Universal Robots PolyScope program: Mycobot.urp

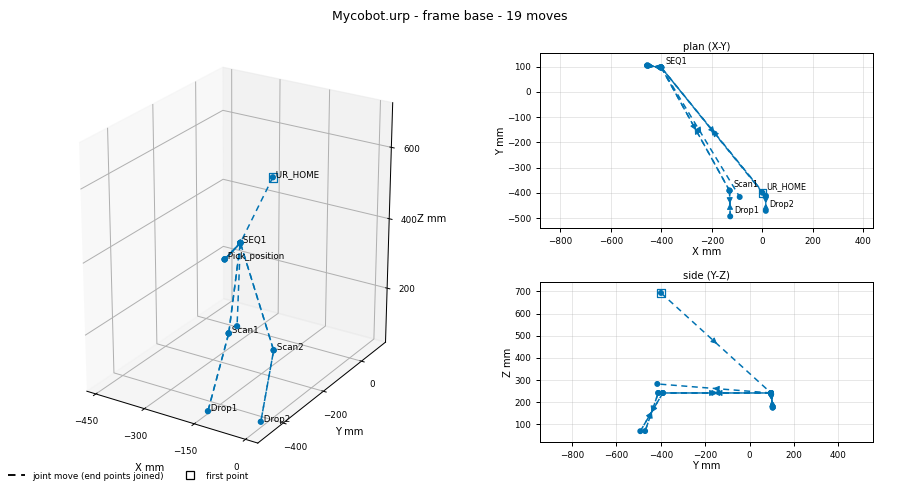
[picture p0: tool path of Mycobot.urp in frame base, 19 of 19 moves have a stored position in this frame; points joined in program order, loops and branches not executed]
Program Mycobot (installation=default directory=/programs createdIn=5.13.0 lastSavedIn=5.13.0 robotSerialNumber=20185300461)
Calibrated DH parameters: a=[-0.000193, -0.207022, -0.182437, 0.000132, -0.000092, 0]; d=[0.151833, 39.901235, 24.993935, -64.763969, 0.085421, 0.09218]; alpha=[1.57101, -0.003228, 0.001706, 1.571505, -1.572476, 0]; deltaTheta=[0, -0.556568, 7.385156, -0.545397, -0.000002, 0]
InitVariablesNode
Robot Program (runOnlyOnce=false)
  MoveJ speed 60 deg/s, acceleration 80 deg/s^2 (useActiveTCP=true) feature=Base
    Waypoint UR_HOME: TCP in base x=0.281 y=-399.322 z=693.096 mm, rx=-0.0014 ry=2.225 rz=-2.2166 rad; joints [-0.001, -90.001, 0, -89.999, 0.001, 0.001] deg; TCP offset x=0 y=0 z=175 mm, rx=0 ry=0 rz=0 rad
    Waypoint SEQ1: TCP in base x=-400.455 y=96.867 z=242.077 mm, rx=-2.2115 ry=-2.1405 rz=0.0251 rad; joints [-173.349, -123.94, -11.31, -131.69, 87.509, 8.47] deg; TCP offset x=0 y=0 z=175 mm, rx=0 ry=0 rz=0 rad
    Wait Sleep waitTime=5
    Waypoint Pick_position: TCP in base x=-456.138 y=104.432 z=176.635 mm, rx=-3.123 ry=0.1229 rz=0.0643 rad; joints [-175.863, -135.405, -11.262, -120.992, 88.708, 98.607] deg
    URCap Gripper (Robotiq_Grippers, Robotiq Inc.) dataModel(position=52.94117647058823, force=36.60130718954249, speed=10.893246187363836, positionInDouble=52.94117647058823, forceInDouble=36.60130718954249, speedInDouble=10.893246187363836, slaveIds=[9], blocking=true, robotCompliant=false)
    URCap Grip Check (Robotiq_Grippers, Robotiq Inc.) dataModel(DimensionKey=100.0, DimensionDimensionPositiveGapKey=5.0, DimensionNegativeGapKey=5.0, GripperIdKey=1, ModelDefinedKey=true, ObjectDetectedKey=true, DimensionValidationKey=false); state(isChildrenLocked=true)
      URCap If (Robotiq_Grippers, Robotiq Inc.)
        Waypoint Waypoint_1: TCP in base x=-400.458 y=96.877 z=242.084 mm, rx=-2.2115 ry=-2.1404 rz=0.0251 rad; joints [-173.351, -123.94, -11.307, -131.691, 87.509, 8.47] deg; TCP offset x=0 y=0 z=175 mm, rx=0 ry=0 rz=0 rad
      URCap Else (Robotiq_Grippers, Robotiq Inc.)
        Wait Sleep waitTime=10
        Popup Message (haltProgram=false message=NO LEGO DETECTED inputType=Text)
    Waypoint Safe_above_pik2: TCP in base x=-400.455 y=96.891 z=242.08 mm, rx=-2.2116 ry=-2.1404 rz=0.0251 rad; joints [-173.353, -123.94, -11.31, -131.689, 87.509, 8.471] deg; TCP offset x=0 y=0 z=175 mm, rx=0 ry=0 rz=0 rad
    Waypoint Scan1: TCP in base x=-130.159 y=-390.915 z=242.077 mm, rx=-0.1811 ry=-3.0992 rz=0.0857 rad; joints [-88.166, -123.94, -11.311, -131.689, 87.507, 8.471] deg; TCP offset x=0 y=0 z=175 mm, rx=0 ry=0 rz=0 rad
    Wait Sleep waitTime=3
    Waypoint Drop1: TCP in base x=-127.488 y=-492.684 z=69.679 mm, rx=-0.1841 ry=-3.0975 rz=0.0473 rad; joints [-88.165, -171.493, 34.819, -131.686, 87.506, 8.471] deg; TCP offset x=0 y=0 z=175 mm, rx=0 ry=0 rz=0 rad
    URCap Gripper (Robotiq_Grippers, Robotiq Inc.) dataModel(position=40.0, force=36.60130718954249, speed=10.893246187363836, positionInDouble=40.0, forceInDouble=36.60130718954249, speedInDouble=10.893246187363836, slaveIds=[9], blocking=true, robotCompliant=false)
    Wait Sleep waitTime=1
    Waypoint Return0: TCP in base x=-130.177 y=-390.911 z=242.06 mm, rx=-0.1811 ry=-3.0991 rz=0.0856 rad; joints [-88.166, -123.941, -11.312, -131.69, 87.503, 8.471] deg; TCP offset x=0 y=0 z=175 mm, rx=0 ry=0 rz=0 rad
    URCap Gripper (Robotiq_Grippers, Robotiq Inc.) dataModel(position=19.607843137254903, force=36.60130718954249, speed=10.893246187363836, positionInDouble=19.607843137254903, forceInDouble=36.60130718954249, speedInDouble=10.893246187363836, slaveIds=[9], blocking=true, robotCompliant=false)
    Waypoint scan01: TCP in base x=-130.136 y=-390.929 z=242.057 mm, rx=-0.1809 ry=-3.0991 rz=0.0856 rad; joints [-88.161, -123.942, -11.311, -131.689, 87.505, 8.47] deg; TCP offset x=0 y=0 z=175 mm, rx=0 ry=0 rz=0 rad
    URCap Gripper (Robotiq_Grippers, Robotiq Inc.) dataModel(position=0.0, force=36.60130718954249, speed=10.893246187363836, positionInDouble=0.0, forceInDouble=36.60130718954249, speedInDouble=10.893246187363836, slaveIds=[9], blocking=true, robotCompliant=false)
    Waypoint SEQ2: TCP in base x=-400.462 y=96.851 z=242.093 mm, rx=-2.2115 ry=-2.1404 rz=0.0252 rad; joints [-173.348, -123.938, -11.309, -131.69, 87.51, 8.472] deg; TCP offset x=0 y=0 z=175 mm, rx=0 ry=0 rz=0 rad
    Wait Sleep waitTime=5
    Waypoint Pickv2: TCP in base x=-456.135 y=104.44 z=176.645 mm, rx=-3.123 ry=0.1229 rz=0.0643 rad; joints [-175.863, -135.404, -11.261, -120.993, 88.707, 98.607] deg; TCP offset x=0 y=0 z=175 mm, rx=0 ry=0 rz=0 rad
    URCap Gripper (Robotiq_Grippers, Robotiq Inc.) dataModel(position=52.94117647058823, force=36.60130718954249, speed=10.893246187363836, positionInDouble=52.94117647058823, forceInDouble=36.60130718954249, speedInDouble=10.893246187363836, slaveIds=[9], blocking=true, robotCompliant=false)
    URCap Grip Check (Robotiq_Grippers, Robotiq Inc.) dataModel(ObjectDetectedKey=true, DimensionValidationKey=false, DimensionKey=100.0, DimensionDimensionPositiveGapKey=5.0, DimensionNegativeGapKey=5.0, GripperIdKey=1, ModelDefinedKey=true); state(isChildrenLocked=true)
      URCap If (Robotiq_Grippers, Robotiq Inc.)
        Waypoint Waypoint_2: TCP in base x=-400.465 y=96.868 z=242.087 mm, rx=-2.2115 ry=-2.1404 rz=0.0252 rad; joints [-173.35, -123.939, -11.31, -131.688, 87.51, 8.469] deg; TCP offset x=0 y=0 z=175 mm, rx=0 ry=0 rz=0 rad
      URCap Else (Robotiq_Grippers, Robotiq Inc.)
        Popup Message (haltProgram=false message=NO LEGO DETECTED inputType=Text)
    Waypoint Scan2: TCP in base x=13.397 y=-411.795 z=242.108 mm, rx=0.3685 ry=-3.0926 rz=0.0947 rad; joints [-67.888, -123.936, -11.31, -131.687, 87.509, 8.47] deg; TCP offset x=0 y=0 z=175 mm, rx=0 ry=0 rz=0 rad
    Wait Sleep waitTime=3
    Waypoint Drop2: motionParameters(nextMotionTime=4); TCP in base x=13.429 y=-470.86 z=70.27 mm, rx=0.1151 ry=-3.0804 rz=-0.1175 rad; joints [-71.076, -136.443, -37.095, -101.486, 88.026, 14.753] deg; TCP offset x=0 y=0 z=175 mm, rx=0 ry=0 rz=0 rad
    URCap Gripper (Robotiq_Grippers, Robotiq Inc.) dataModel(position=20.0, force=36.60130718954249, speed=5.893246187363836, positionInDouble=20.0, forceInDouble=36.60130718954249, speedInDouble=5.893246187363836, slaveIds=[9], blocking=true, robotCompliant=false)
    Wait Sleep waitTime=1
    Waypoint return2: TCP in base x=13.376 y=-411.788 z=242.115 mm, rx=0.3685 ry=-3.0926 rz=0.0947 rad; joints [-67.89, -123.934, -11.31, -131.689, 87.508, 8.47] deg; TCP offset x=0 y=0 z=175 mm, rx=0 ry=0 rz=0 rad
    URCap Gripper (Robotiq_Grippers, Robotiq Inc.) dataModel(position=0.0, force=36.60130718954249, speed=10.893246187363836, positionInDouble=0.0, forceInDouble=36.60130718954249, speedInDouble=10.893246187363836, slaveIds=[9], blocking=true, robotCompliant=false)
    Waypoint SEQ3: TCP in base x=-400.453 y=96.873 z=242.086 mm, rx=-2.2114 ry=-2.1405 rz=0.0251 rad; joints [-173.349, -123.938, -11.312, -131.69, 87.508, 8.469] deg; TCP offset x=0 y=0 z=175 mm, rx=0 ry=0 rz=0 rad
    Wait Sleep waitTime=5
    Waypoint Pick3: TCP in base x=-456.124 y=104.431 z=176.641 mm, rx=-3.123 ry=0.1229 rz=0.0643 rad; joints [-175.862, -135.403, -11.262, -120.996, 88.707, 98.609] deg; TCP offset x=0 y=0 z=175 mm, rx=0 ry=0 rz=0 rad
    URCap Gripper (Robotiq_Grippers, Robotiq Inc.) dataModel(position=67.45098039215686, force=39.60130718954249, speed=10.893246187363836, positionInDouble=67.45098039215686, forceInDouble=39.60130718954249, speedInDouble=10.893246187363836, slaveIds=[9], blocking=true, robotCompliant=false)
    URCap Grip Check (Robotiq_Grippers, Robotiq Inc.) dataModel(ObjectDetectedKey=true, DimensionValidationKey=false, DimensionKey=100.0, DimensionDimensionPositiveGapKey=5.0, DimensionNegativeGapKey=5.0, GripperIdKey=1, ModelDefinedKey=true); state(isChildrenLocked=true)
      URCap If (Robotiq_Grippers, Robotiq Inc.)
        Waypoint Waypoint_3: TCP in base x=-400.472 y=96.852 z=242.093 mm, rx=-2.2114 ry=-2.1405 rz=0.0252 rad; joints [-173.347, -123.939, -11.309, -131.688, 87.509, 8.469] deg; TCP offset x=0 y=0 z=175 mm, rx=0 ry=0 rz=0 rad
      URCap Else (Robotiq_Grippers, Robotiq Inc.)
        Popup Message (haltProgram=false message=NO LEGO DETECTED inputType=Text)
    Waypoint Scan3: TCP in base x=-89.876 y=-415.99 z=282.749 mm, rx=-0.0363 ry=-3.1126 rz=0.3325 rad; joints [-82.601, -123.939, -2.285, -131.689, 87.511, 8.469] deg; TCP offset x=0 y=0 z=175 mm, rx=0 ry=0 rz=0 rad
    Wait Sleep waitTime=3
